// Gets the upper bound index of the array of specified type.
FUNCTION F_GetIntArrayUpperBound : T_Position // The upper bound index of the specified array.
VAR_IN_OUT
	arArray : ARRAY[*] OF INT; // The array to query.
END_VAR

F_GetIntArrayUpperBound := UPPER_BOUND(arArray, 1);

END_FUNCTION

(* stored: Version 1.1.0.1
   POU F_GetIntArrayUpperBound: Id {1d69981d-c0d5-0299-3207-c458c92277b1}, SpecialFunc None *)
